// TIA Portal V20 export
VAR_GLOBAL   // PLC tag table "Default tag table"
   System_Byte AT %MB1 : Byte;
   FirstScan AT %M1.0 : Bool;
   DiagStatusUpdate AT %M1.1 : Bool;
   AlwaysTRUE AT %M1.2 : Bool;
   AlwaysFALSE AT %M1.3 : Bool;
   Clock_Byte AT %MB0 : Byte;
   Clock_10Hz AT %M0.0 : Bool;
   Clock_5Hz AT %M0.1 : Bool;
   "Clock_2.5Hz" AT %M0.2 : Bool;
   Clock_2Hz AT %M0.3 : Bool;
   "Clock_1.25Hz" AT %M0.4 : Bool;
   Clock_1Hz AT %M0.5 : Bool;
   "Clock_0.625Hz" AT %M0.6 : Bool;
   "Clock_0.5Hz" AT %M0.7 : Bool;
   Tag_1 AT %M99.0 : Bool;
   Tag_2 AT %MD1000 : DWord;
   Tag_3 AT %MW20 : Word;
   Tag_4 AT %MW40 : Word;
   Tag_5 AT %MW42 : Word;
   Tag_6 AT %MW44 : Word;
   Tag_7 AT %MW100 : Word;
   Tag_8 AT %MW102 : Word;
   Tag_9 AT %MW104 : Word;
   Tag_10 AT %MD150 : DWord;
END_VAR
